// TIA Portal V21 export
TYPE "Std_StrutturaRicetta_Spiedinatrice"
   STRUCT
      NomeFormato : String[20];   // p01
      QuotaPrimoInserimentoStecchi : Real;   // p07
      DistanzaTraGliStecchi : Real;   // p04
      NumeroFilePerLato : DInt;   // p03
      QuoteFileStecchiNelCubo : Array[0..30] of Real;
      LunghezzaStecco : Real;   // p06
      LarghezzaStecco : Real;   // p05
      NumeroStecchi : DInt;   // p02
      AltezzaTotCubo : DInt;   // p08
      NumeroCicliTaglio : DInt;
   END_STRUCT;
END_TYPE
